// This function has been automatically generated from the project information.
{attribute 'signature_flag' := '1073741824'}
{attribute 'TcGenerated'}
{attribute 'no-analysis'}
FUNCTION F_GetCompany : WSTRING
VAR_INPUT
	
END_VAR

F_GetCompany := "TcHaxx";

END_FUNCTION

(* stored: Version 1.1.0.1
   POU F_GetCompany: Id {ea569029-20e1-4427-8402-25df751484e6}, SpecialFunc None *)
